// TIA Portal V18 export
TYPE "ST_KeyenceSR1000"
// stored: IsFailsafeCompliant false
   STRUCT
      Common : Struct   // 通用变量
         nMode : Int;   // 模式
         bError : Bool;   // 错误
         bWarning : Bool;   // 警告
         bReset : Bool;   // 复位按钮
         bDone : Bool;   // 完成信号
         bOK : Bool;
         bNG : Bool;
         bScreenActive : Bool;   // 屏幕激活
         nErrorNo : Int;   // 错误代码
         nWarningNo : Int;   // 警告代码
      END_STRUCT;
      In : Struct
         bError : Bool;   // 报警中
         bBusy : Bool;
         bReadComplete : Bool;   // 读取完成
         bReadFailure : Bool;   // 读取失败
         nReadResultCode : Int;   // 错误代码
         nDataSize : UInt;   // 数据长度
         aData : Array[1..128] of Char;   // 结果数据输出
      END_STRUCT;
      Out : Struct
         bErrorClear : Bool;   // 报警清除
         bReadRequest : Bool;   // 开始读取
         bReadComlpleteClear : Bool;   // 读取完成清除
      END_STRUCT;
      Pare : Struct
         tMaxProcessTime : Time := T#10S;
      END_STRUCT;
      RecordCode : String[128];   // 结果数据
   END_STRUCT;
END_TYPE
